{attribute 'linkalways'} 
{attribute 'no_explicit_call' := 'This FB is a CLASS and must be accessed using methods or properties'}
{attribute 'enable_dynamic_creation'}
FUNCTION_BLOCK Node_F_VN_LineIntersectionPoint EXTENDS VisionNode
VAR
    aLine1 : _TcVnVector4_LREAL;
    aLine2 : _TcVnVector4_LREAL;
    aIntersecPoint : _TcVnPoint2_REAL;
    hrPrev : _HRESULT(S_OK);
	hresult : _HRESULT(S_OK);
END_VAR

METHOD PUBLIC  Clone : I_Node
VAR
	pNode : POINTER TO Node_F_VN_LineIntersectionPoint;
END_VAR
pNode := __NEW(Node_F_VN_LineIntersectionPoint);
Clone := pNode^;
END_METHOD

METHOD FB_init : BOOL
VAR_INPUT
	bInitRetains : BOOL; // if TRUE, the retain variables are initialized (warm start / cold start)
	bInCopyCode : BOOL;  // if TRUE, the instance afterwards gets moved into the copy code (online change)
END_VAR
AddInput('aLine1', aLine1);
AddInput('aLine2', aLine2);
AddInput('hrPrev', hrPrev);
AddOutput('aIntersecPoint', aIntersecPoint);
AddOutput('hresult',hresult);
END_METHOD

METHOD PROTECTED OnExecute
hresult.Value := F_VN_LineIntersectionPoint(
	aLine1 := aLine1.Value,
    aLine2 := aLine2.Value,
    aIntersecPoint := aIntersecPoint.Value,
	hrPrev:= hrPrev.Value);
END_METHOD

METHOD PUBLIC PreExecutionCheck
VAR_INPUT
	Check : I_PreExecutionChecks;
END_VAR
END_METHOD

END_FUNCTION_BLOCK

(* stored: Version 1.1.0.1, ProductVersion 3.1.4024.13
   POU Node_F_VN_LineIntersectionPoint: Id {bf6ec5b5-cbf2-08fc-0bbc-e7ff62559348}, SpecialFunc None
   Folder Constructor: Id {53a900da-c7d7-0e6f-317e-ba10c144b301}
   Method Clone: Id {95e522fc-45ce-0ed6-0cba-0eea2012a5f9}
   Method FB_init: Id {268b8206-007d-072c-237c-154b44921bf7}
   Method OnExecute: Id {673922be-baa2-093f-161a-1943385b69e6}
   Method PreExecutionCheck: Id {e521388b-f6d9-006b-0ae8-22701470c413} *)
